// TwinCAT 3 PLC project Untitled1
// ProgramVersion: 3.1.4026.19
// libraries:
//   Tc2_Standard, * (Beckhoff Automation GmbH)
//   Tc2_System, * (Beckhoff Automation GmbH)
// project tree:
//   / PlcTask.TcTTO
//   POUs/ uloha1.TcPOU, uloha2.TcPOU
// real-time tasks:
//   TASK PlcTask: cycle T#10ms, priority 20, ADS port 350

CONFIGURATION Untitled1
    RESOURCE PLC ON TwinCAT3
        TASK PlcTask(INTERVAL := T#10ms, PRIORITY := 20);
        PROGRAM uloha2 WITH PlcTask : uloha2;
        PROGRAM uloha1 WITH PlcTask : uloha1;
    END_RESOURCE
END_CONFIGURATION

// ---- POUs/uloha2.TcPOU
PROGRAM uloha2
VAR
	stop3: BOOL;
	stop2: BOOL;
	stop1: BOOL;
	M1: BOOL;
	M2: BOOL;
	M3: BOOL;
	start1: BOOL;
	start2: BOOL;
	start3: BOOL;
	stav: INT;
	pocet_motorov: INT;
	stop: BOOL;
END_VAR

pocet_motorov := 0;

IF M1 THEN pocet_motorov := pocet_motorov + 1; END_IF;
IF M2 THEN pocet_motorov := pocet_motorov + 1; END_IF;
IF M3 THEN pocet_motorov := pocet_motorov + 1; END_IF;


IF stop1 THEN
    M1 := FALSE;
    start1 := FALSE;
    stop1 := FALSE;
END_IF;

IF stop2 THEN
    M2 := FALSE;
    start2 := FALSE;
    stop2 := FALSE;
END_IF;

IF stop3 THEN
    M3 := FALSE;
    start3 := FALSE;
    stop3 := FALSE;
END_IF;



CASE stav OF

    0:
        IF start1 THEN
            M1 := TRUE;
            stav := 1;
        ELSIF start2 THEN
            M2 := TRUE;
            stav := 1;
        ELSIF start3 THEN
            M3 := TRUE;
            stav := 1;
        END_IF;

    1:
        IF pocet_motorov >= 2 THEN
            stav := 2;
        ELSE
            IF start1 AND (NOT M1) THEN M1 := TRUE; END_IF;
            IF start2 AND (NOT M2) THEN M2 := TRUE; END_IF;
            IF start3 AND (NOT M3) THEN M3 := TRUE; END_IF;
        END_IF;

    2:
        IF pocet_motorov < 2 THEN
            stav := 1;
        END_IF;

END_CASE;


IF stop THEN
    M1 := FALSE;
    M2 := FALSE;
    M3 := FALSE;

    pocet_motorov := 0;
    stav := 0;

    start1 := FALSE;
    start2 := FALSE;
    start3 := FALSE;

    stop1 := FALSE;
    stop2 := FALSE;
    stop3 := FALSE;

    stop := FALSE;
END_IF;

END_PROGRAM

// ---- POUs/uloha1.TcPOU
PROGRAM uloha1
VAR
	stop: bool;
	Motor: bool;
	start: bool;
	stav: INT;
	casovac: TON;
	casovac2: Ton;
	RUN: BOOL;
	stopDelay: Ton;
	resetDelay: ton;
END_VAR


IF stop THEN
    RUN := FALSE;

ELSIF start THEN
    RUN := TRUE;
END_IF;

CASE stav OF

    0: 
        Motor := FALSE;
        casovac(IN := FALSE, PT := T#5S);

        IF RUN THEN
            stav := 10;
        END_IF;


    10: 
        Motor := TRUE;
        casovac(IN := TRUE, PT := T#5S);

        IF casovac.Q THEN
            casovac(IN := FALSE, PT := T#5S);  
            stav := 20;
        END_IF;

        IF NOT RUN THEN
            stav := 0;
        END_IF;

    20: 
        Motor := FALSE;
        casovac(IN := TRUE, PT := T#5S);

        IF casovac.Q THEN
            casovac(IN := FALSE, PT := T#5S);   
            stav := 10;
        END_IF;

        IF NOT RUN THEN
            stav := 0;
        END_IF;

END_CASE;
IF stop = TRUE THEN
    resetDelay(IN := TRUE, PT := T#1S);
END_IF;

IF resetDelay.Q THEN
    Motor := FALSE;
    start := FALSE;
    stop := FALSE;        
    resetDelay(IN := FALSE, PT := T#1S);
END_IF;

END_PROGRAM
